// TIA Portal V16 export
// export: Created 2021-05-25T16:14:41.3201809Z, ExportSetting WithDefaults, DisplayName Totally Integrated Automation Portal, DisplayVersion V16, DisplayName TIA Portal Version Control Interface, DisplayVersion V16, DisplayName TIA Portal Openness, DisplayVersion V16, DisplayName STEP 7 Professional, DisplayVersion V16, DisplayName STEP 7 Safety, DisplayVersion V16, DisplayName WinCC Unified SCADA Engineering System, DisplayVersion V16
DATA_BLOCK "dbOPAlarms"   // DB112
{ S7_Optimized_Access := 'FALSE'; DB_Accessible_From_OPC_UA := 'FALSE' }
VERSION : 0.1
// stored: AutoNumber false, DBAccessibleFromOPCUA false, IsOnlyStoredInLoadMemory false, IsWriteProtectedInAS false
   VAR
      Alarm : Array[0..63] of Bool;   // System Alarms
      OPAlarmWord : Array[0..3] of Word;   // OP Alarms
      AlarmACK : Array[0..63] of Bool;
   END_VAR
BEGIN
END_DATA_BLOCK
